TYPE AX5000_P_0851 :
STRUCT
	Save_amplifier_identification:UINT;
END_STRUCT
END_TYPE

(* stored: Version 1.1.0.1, ProductVersion 3.1.4024.3
   DUT AX5000_P_0851: Id {d84eccb2-b29d-44c5-8435-7680d17edd61} *)
